{attribute 'qualified_only'}
VAR_GLOBAL
	mb_Input_Coils:ARRAY[0..255] OF BOOL;
	mb_Output_Coils:ARRAY[0..255] OF BOOL;
	mb_Output_Registers:ARRAY[0..2000] OF DINT;
	mb_Input_Registers:ARRAY[0..2000] OF WORD;	
END_VAR

(* stored: Version 1.1.0.1, ProductVersion 3.1.4024.6
   GVL GVL_MB: Id {76e83e92-525f-4e7c-8225-8eea945b5bf4} *)
